// TIA Portal V20 export
FUNCTION_BLOCK "LER_LaserMark"   // FB9, LAD
// stored: Access Published, MemoryReserve 100, SetENOAutomatically false
   VAR_INPUT
      enable : Bool;
      enableManualCmds : Bool;
      jellyRollUsed : Bool;   // Unused is dryrun, gaugeRnR etc..
      simulationCmds : Bool;
      errAckHmi : Bool;
      interlock : Bool;
      autoGenMarkingData : String[32];
   END_VAR
   VAR_OUTPUT
      lagerMarkingTrigger : Bool;
      error : Bool;
      errorCode : Word;
   END_VAR
   VAR_IN_OUT
      configuration : "LER_typeLaserMarkConfiguration";
      moduleInterface : "LER_typeLaserMarkInterface";
      controlNode : "LER_typeLaserMarkControlNode";
   END_VAR
   VAR
      instTONTimer { S7_SetPoint := 'True'} : Array[0..19] of IEC_TIMER;
      statCmd { ExternalAccessible := 'False'; ExternalVisible := 'False'; ExternalWritable := 'False'} : "LER_typeLaserMarkCommands";
      statMonitoring { ExternalAccessible := 'False'; ExternalVisible := 'False'; ExternalWritable := 'False'} : "LER_typeLaserMarkMonitoring";
      statConfig { ExternalAccessible := 'False'; ExternalVisible := 'False'; ExternalWritable := 'False'} : "LER_typeLaserMarkConfiguration";
      statRetValInt { ExternalAccessible := 'False'; ExternalVisible := 'False'; ExternalWritable := 'False'} : Array[1..#count] of Int;
      statRetValWord { ExternalAccessible := 'False'; ExternalVisible := 'False'; ExternalWritable := 'False'} : Array[1..#count] of Word;
      statBit { ExternalAccessible := 'False'; ExternalVisible := 'False'; ExternalWritable := 'False'} : Array[0..49] of Bool;
      statAction { ExternalAccessible := 'False'; ExternalVisible := 'False'; ExternalWritable := 'False'} : Array[0..49] of Bool;
      statOutputCharData { ExternalAccessible := 'False'; ExternalVisible := 'False'; ExternalWritable := 'False'} : Array[1..128] of Char;
      statTpTimer { S7_SetPoint := 'True'} : Array[0..1] of TP_TIME;
      statPulse : Array[0..999] of Bool;
      statTonTimer { S7_SetPoint := 'True'} : Array[0..999] of TON_TIME;
      statProgramChange : Array[0..999] of Bool;
      "step" { ExternalAccessible := 'False'; ExternalVisible := 'False'; ExternalWritable := 'False'} : Int;
      statHold : Bool;
   END_VAR
   VAR_TEMP
      tempRetVal : Array[1..#count] of Int;
      tempCnt : Array[0..9] of UInt;
      tempCharDataDelete : Array[1..128] of Char;
      tempStringDataDelete : String[128];
      tempProgramNoDelete : DWord;
      tempIndex : Int;
   END_VAR
   VAR CONSTANT
      delayTime : Time := T#2s;
      count : Int := 16;
      statusNoErrorOccurred : Word := 16#0000;   // No error occurred.
      errMachine : Word := 16#8000;
      errRequest : Word := 16#8001;
      errHwdNotConfigured : Word := 16#8090;   // You have not configured a module for the specified hardware identifier or You have ignored the restriction concerning the length of consistent data, or you have not specified a hardware identifier as an address at parameter LADDR
      errRecordDataType : Word := 16#8092;   // Non-supported data type in the RECORD parameter.
      errNoDpProfinetIoModule : Word := 16#8093;   // No DP module/PROFINET IO device from which you can read consistent data exists for the hardware identifier specified in LADDR . This error code also occurs if the module addressed by means of LADDR does not have inputs.
      errIoAccessPermission : Word := 16#80A0;   // An access error was detected when accessing the I/O.
      errRecordLengthInsufficient : Word := 16#80B1;   // The length of the specified destination area at parameter RECORD is shorter than the configured user data length.
      errDataNotReceived : Word := 16#80C0;   // The data have not been read yet.
   END_VAR
   // // statBit[0] : data setting
   // // statBit[1] : delete data move
   // // statBit[2] : set data save
   // // statBit[3] : data write done
   // // statBit[4] : data writing
   // // statBit[5] : CMD_saveBT
   // // statBit[6] : CMD_save interlock
   // // statBit[7] : sequence hold
   // // statBit[8] : ( Not empty data ) read data save
   // // statBit[9] : ( Empty data ) read data save
   // // statBit[10] : write String To Char
   // // statBit[11] : done String To Char
   // // statBit[12] : P Trig
   // // statBit[15] : Temp config Save
   // // statBit[16] : config Save Lock
   // // statBit[17] : config Save Writing
   // // statBit[25] : trigger
   VAR_TEMP   // added for the SCL form of the ladder/FBD networks
      _w1 : Bool;
      _w2 : Bool;
      _w3 : Bool;
      _w4 : Bool;
      _w5 : Bool;
      _w6 : Bool;
      _w7 : Bool;
      _w8 : Bool;
      _w9 : Bool;
   END_VAR
BEGIN

REGION Network 1 (SCL): DP READ
   REGION DP read

       IF #enable AND NOT #simulationCmds THEN
           #"statRetValInt"[1] := DPRD_DAT(LADDR := #configuration.hwID.machineStatusID, RECORD => #statMonitoring.profinetInput.machineStatus);
           #"statRetValInt"[2] := DPRD_DAT(LADDR := #configuration.hwID.functionStatusID, RECORD => #statMonitoring.profinetInput.functionStatus);
           #"statRetValInt"[3] := DPRD_DAT(LADDR := #configuration.hwID.completionStatusID, RECORD => #statMonitoring.profinetInput.completionStatus);
           #"statRetValInt"[4] := DPRD_DAT(LADDR := #configuration.hwID.errorStatusID, RECORD => #statMonitoring.profinetInput.errorStatus);
           #"statRetValInt"[5] := DPRD_DAT(LADDR := #configuration.hwID.errorCodesID, RECORD => #statMonitoring.profinetInput.errorCodes);
           #"statRetValInt"[6] := DPRD_DAT(LADDR := #configuration.hwID.operateParameterID, RECORD => #statMonitoring.profinetInput.operateParameter);
           #"statRetValInt"[7] := DPRD_DAT(LADDR := #configuration.hwID."2DCReadResultID", RECORD => #statMonitoring.profinetInput."2DCReadResult");
           #"statRetValInt"[8] := DPRD_DAT(LADDR := #configuration.hwID.countResultDataID, RECORD => #statMonitoring.profinetInput.countResultData);
           #"statRetValInt"[9] := DPRD_DAT(LADDR := #configuration.hwID.resultDataID, RECORD => #statMonitoring.profinetInput.resultData);
       END_IF;

   END_REGION
END_REGION

REGION Network 2 (SCL): INPUT MAPPING
   REGION Input mapping

       IF #enable THEN
           // Command
           IF #enableManualCmds THEN
               #statCmd.start := #moduleInterface.commands.start;
               #statCmd.configSave := #moduleInterface.commands.configSave;
               #statMonitoring.profinetOutput.generalRequest.guideLaserRequest := #moduleInterface.commands.guideRequest;
               #statConfig.markingProgramNo := #moduleInterface.configuration.markingProgramNo;
           ELSE
               #statCmd.start := #controlNode.commands.start;
               #statCmd.configSave := #controlNode.commands.configSave;
               #statMonitoring.profinetOutput.generalRequest.guideLaserRequest := #controlNode.commands.guideRequest;
               #statConfig.markingProgramNo := #configuration.markingProgramNo;
           END_IF;

           #statCmd.generateMode := #moduleInterface.commands.generateMode;

           IF #statCmd.generateMode THEN
               #statConfig.markingData := #autoGenMarkingData;
           ELSE
               #statConfig.markingData := #moduleInterface.configuration.markingData;
           END_IF;

           #statMonitoring.data := #statConfig.markingData;

           #statMonitoring.error := #statMonitoring.profinetInput.machineStatus.errorStatus;
           #statMonitoring.warning := #statMonitoring.profinetInput.machineStatus.warningStatus;
           #statMonitoring.errorCode := #errorCode;

       END_IF;

   END_REGION
END_REGION

REGION Network 3 (SCL): ERROR STATUS
   REGION Error check

       IF #enable AND NOT #simulationCmds THEN
           IF #statRetValInt <> #tempRetVal THEN
               FOR #tempIndex := 1 TO #count DO
                   #statRetValWord[#tempIndex] := INT_TO_WORD(#statRetValInt[#tempIndex]); // convert the return value of DPRD, DPWR form int to word
                   CASE #statRetValWord[#tempIndex] OF

                       #errHwdNotConfigured:
                           #errorCode := #errHwdNotConfigured;

                       #errRecordDataType:
                           #errorCode := #errRecordDataType;

                       #errNoDpProfinetIoModule:
                           #errorCode := #errNoDpProfinetIoModule;

                       #errIoAccessPermission:
                           #errorCode := #errIoAccessPermission;

                       #errRecordLengthInsufficient:
                           #errorCode := #errRecordLengthInsufficient;

                       #errDataNotReceived:
                           #errorCode := #errDataNotReceived;
                   END_CASE;
               END_FOR;

           ELSIF #statMonitoring.profinetInput.machineStatus.errorStatus THEN
               #errorCode := #errMachine;

           ELSIF #statMonitoring.profinetInput.errorStatus.startMarkingRequestError OR
               #statMonitoring.profinetInput.errorStatus.stopMarkingRequestError OR
               #statMonitoring.profinetInput.errorStatus.errorClearRequestError OR
               #statMonitoring.profinetInput.errorStatus."2DCReadRequestError" OR
               #statMonitoring.profinetInput.errorStatus.commandSendRequestError THEN
               #errorCode := #errRequest;

           ELSE
               #errorCode := #statusNoErrorOccurred;
           END_IF;
       ELSE
           #errorCode := #statusNoErrorOccurred;
       END_IF;

       #error := #errorCode <> 0;

   END_REGION
END_REGION

REGION Network 4: ERROR ACK
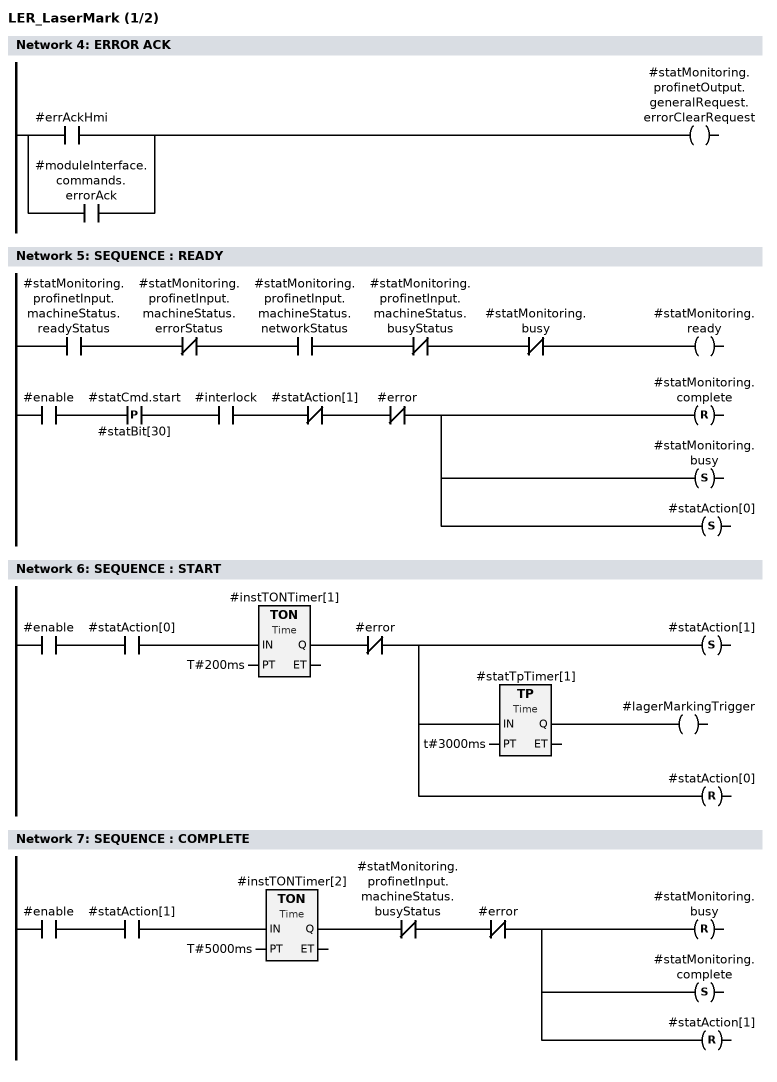
   RUNG wire#powerrail
      Contact( #errAckHmi )
      wire#w1
      Coil( #statMonitoring.profinetOutput.generalRequest.errorClearRequest )
   END_RUNG
   RUNG wire#powerrail
      Contact( #moduleInterface.commands.errorAck )
   END_RUNG wire#w1
   // the same network as SCL:
   #statMonitoring.profinetOutput.generalRequest.errorClearRequest := #errAckHmi OR #moduleInterface.commands.errorAck;
END_REGION

REGION Network 5: SEQUENCE : READY
   RUNG wire#powerrail
      Contact( #statMonitoring.profinetInput.machineStatus.readyStatus )
      I_Contact( #statMonitoring.profinetInput.machineStatus.errorStatus )
      Contact( #statMonitoring.profinetInput.machineStatus.networkStatus )
      I_Contact( #statMonitoring.profinetInput.machineStatus.busyStatus )
      I_Contact( #statMonitoring.busy )
      Coil( #statMonitoring.ready )
   END_RUNG
   RUNG wire#powerrail
      Contact( #enable )
      P_Contact(operand := #statCmd.start, bit := #statBit[30])
      Contact( #interlock )
      I_Contact( #statAction[1] )
      I_Contact( #error )
      wire#w1
      R_Coil( #statMonitoring.complete )
   END_RUNG
   RUNG wire#w1
      S_Coil( #statMonitoring.busy )
   END_RUNG
   RUNG wire#w1
      S_Coil( #statAction[0] )
   END_RUNG
   // the same network as SCL:
   #statMonitoring.ready := #statMonitoring.profinetInput.machineStatus.readyStatus AND NOT #statMonitoring.profinetInput.machineStatus.errorStatus AND #statMonitoring.profinetInput.machineStatus.networkStatus AND NOT #statMonitoring.profinetInput.machineStatus.busyStatus AND NOT #statMonitoring.busy;
   #_w1 := #enable AND #statCmd.start AND NOT #statBit[30];   // rising edge of #statCmd.start
   #statBit[30] := #statCmd.start;
   IF #_w1 AND #interlock AND NOT #statAction[1] AND NOT #error THEN
       #statMonitoring.complete := FALSE;
       #statMonitoring.busy := TRUE;
       #statAction[0] := TRUE;
   END_IF;
END_REGION

REGION Network 6: SEQUENCE : START
   RUNG wire#powerrail
      Contact( #enable )
      Contact( #statAction[0] )
      { S7_Templates := "time_type := Time" } #instTONTimer[1].TON(pt := T#200ms, et =>)
      I_Contact( #error )
      wire#w1
      S_Coil( #statAction[1] )
   END_RUNG
   RUNG wire#w1
      { S7_Templates := "time_type := Time" } #statTpTimer[1].TP(pt := t#3000ms, et =>)
      Coil( #lagerMarkingTrigger )
   END_RUNG
   RUNG wire#w1
      R_Coil( #statAction[0] )
   END_RUNG
   // the same network as SCL:
   #instTONTimer[1].TON(IN := #enable AND #statAction[0], PT := T#200ms);
   #_w1 := #instTONTimer[1].Q AND NOT #error;
   IF #_w1 THEN #statAction[1] := TRUE; END_IF;
   #statTpTimer[1].TP(IN := #_w1, PT := t#3000ms);
   #lagerMarkingTrigger := #statTpTimer[1].Q;
   IF #_w1 THEN #statAction[0] := FALSE; END_IF;
END_REGION

REGION Network 7: SEQUENCE : COMPLETE
   RUNG wire#powerrail
      Contact( #enable )
      Contact( #statAction[1] )
      { S7_Templates := "time_type := Time" } #instTONTimer[2].TON(pt := T#5000ms, et =>)
      I_Contact( #statMonitoring.profinetInput.machineStatus.busyStatus )
      I_Contact( #error )
      wire#w1
      R_Coil( #statMonitoring.busy )
   END_RUNG
   RUNG wire#w1
      S_Coil( #statMonitoring.complete )
   END_RUNG
   RUNG wire#w1
      R_Coil( #statAction[1] )
   END_RUNG
   // the same network as SCL:
   #instTONTimer[2].TON(IN := #enable AND #statAction[1], PT := T#5000ms);
   IF #instTONTimer[2].Q AND NOT #statMonitoring.profinetInput.machineStatus.busyStatus AND NOT #error THEN
       #statMonitoring.busy := FALSE;
       #statMonitoring.complete := TRUE;
       #statAction[1] := FALSE;
   END_IF;
END_REGION

REGION Network 8: CONFIGURATION
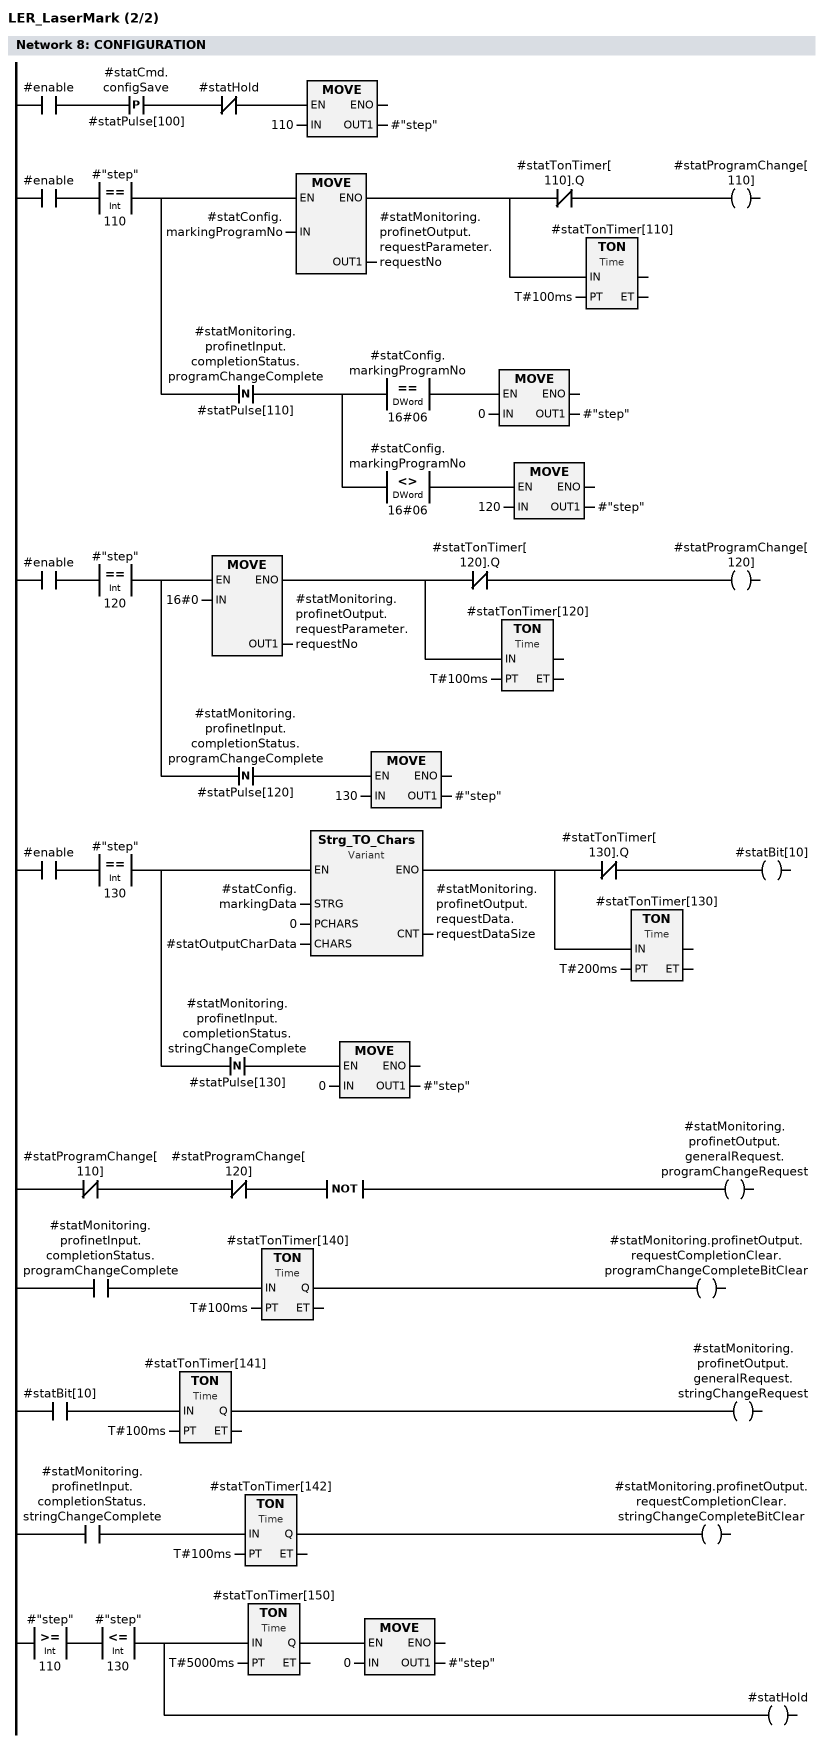
   RUNG wire#powerrail
      Contact( #enable )
      P_Contact(operand := #statCmd.configSave, bit := #statPulse[100])
      I_Contact( #statHold )
      Move(in := 110, out1 => #"step")
   END_RUNG
   RUNG wire#powerrail
      Contact( #enable )
      { S7_Templates := "SrcType := Int" } EQ_Contact(in1 := #"step", in2 := 110)
      wire#w1
      Move(in := #statConfig.markingProgramNo, out1 => #statMonitoring.profinetOutput.requestParameter.requestNo)
      wire#w2
      I_Contact( #statTonTimer[110].Q )
      Coil( #statProgramChange[110] )
   END_RUNG
   RUNG wire#w2
      { S7_Templates := "time_type := Time" } #statTonTimer[110].TON(pt := T#100ms, et =>)
   END_RUNG
   RUNG wire#w1
      N_Contact(operand := #statMonitoring.profinetInput.completionStatus.programChangeComplete, bit := #statPulse[110])
      wire#w3
      { S7_Templates := "SrcType := DWord" } EQ_Contact(in1 := #statConfig.markingProgramNo, in2 := 16#06)
      Move(in := 0, out1 => #"step")
   END_RUNG
   RUNG wire#w3
      { S7_Templates := "SrcType := DWord" } NE_Contact(in1 := #statConfig.markingProgramNo, in2 := 16#06)
      Move(in := 120, out1 => #"step")
   END_RUNG
   RUNG wire#powerrail
      Contact( #enable )
      { S7_Templates := "SrcType := Int" } EQ_Contact(in1 := #"step", in2 := 120)
      wire#w4
      Move(in := 16#0, out1 => #statMonitoring.profinetOutput.requestParameter.requestNo)
      wire#w5
      I_Contact( #statTonTimer[120].Q )
      Coil( #statProgramChange[120] )
   END_RUNG
   RUNG wire#w5
      { S7_Templates := "time_type := Time" } #statTonTimer[120].TON(pt := T#100ms, et =>)
   END_RUNG
   RUNG wire#w4
      N_Contact(operand := #statMonitoring.profinetInput.completionStatus.programChangeComplete, bit := #statPulse[120])
      Move(in := 130, out1 => #"step")
   END_RUNG
   RUNG wire#powerrail
      Contact( #enable )
      { S7_Templates := "SrcType := Int" } EQ_Contact(in1 := #"step", in2 := 130)
      wire#w6
      { S7_Templates := "[ptr_type := Variant, strg_type := String]" } Strg_TO_Chars(Strg := #statConfig.markingData, pChars := 0, Chars := #statOutputCharData, Cnt => #statMonitoring.profinetOutput.requestData.requestDataSize)
      wire#w7
      I_Contact( #statTonTimer[130].Q )
      Coil( #statBit[10] )
   END_RUNG
   RUNG wire#w7
      { S7_Templates := "time_type := Time" } #statTonTimer[130].TON(pt := T#200ms, et =>)
   END_RUNG
   RUNG wire#w6
      N_Contact(operand := #statMonitoring.profinetInput.completionStatus.stringChangeComplete, bit := #statPulse[130])
      Move(in := 0, out1 => #"step")
   END_RUNG
   RUNG wire#powerrail
      I_Contact( #statProgramChange[110] )
      I_Contact( #statProgramChange[120] )
      Not()
      Coil( #statMonitoring.profinetOutput.generalRequest.programChangeRequest )
   END_RUNG
   RUNG wire#powerrail
      Contact( #statMonitoring.profinetInput.completionStatus.programChangeComplete )
      { S7_Templates := "time_type := Time" } #statTonTimer[140].TON(pt := T#100ms, et =>)
      Coil( #statMonitoring.profinetOutput.requestCompletionClear.programChangeCompleteBitClear )
   END_RUNG
   RUNG wire#powerrail
      Contact( #statBit[10] )
      { S7_Templates := "time_type := Time" } #statTonTimer[141].TON(pt := T#100ms, et =>)
      Coil( #statMonitoring.profinetOutput.generalRequest.stringChangeRequest )
   END_RUNG
   RUNG wire#powerrail
      Contact( #statMonitoring.profinetInput.completionStatus.stringChangeComplete )
      { S7_Templates := "time_type := Time" } #statTonTimer[142].TON(pt := T#100ms, et =>)
      Coil( #statMonitoring.profinetOutput.requestCompletionClear.stringChangeCompleteBitClear )
   END_RUNG
   RUNG wire#powerrail
      { S7_Templates := "SrcType := Int" } GE_Contact(in1 := #"step", in2 := 110)
      { S7_Templates := "SrcType := Int" } LE_Contact(in1 := #"step", in2 := 130)
      wire#w8
      { S7_Templates := "time_type := Time" } #statTonTimer[150].TON(pt := T#5000ms, et =>)
      Move(in := 0, out1 => #"step")
   END_RUNG
   RUNG wire#w8
      Coil( #statHold )
   END_RUNG
   // the same network as SCL:
   #_w1 := #enable AND #statCmd.configSave AND NOT #statPulse[100];   // rising edge of #statCmd.configSave
   #statPulse[100] := #statCmd.configSave;
   IF #_w1 AND NOT #statHold THEN #"step" := 110; END_IF;
   #_w2 := #enable AND (#"step" = 110);
   IF #_w2 THEN
       #statMonitoring.profinetOutput.requestParameter.requestNo := #statConfig.markingProgramNo;
   END_IF;
   #statProgramChange[110] := #_w2 AND NOT #statTonTimer[110].Q;
   #statTonTimer[110].TON(IN := #_w2, PT := T#100ms);
   #_w3 := #_w2 AND NOT #statMonitoring.profinetInput.completionStatus.programChangeComplete AND #statPulse[110];   // falling edge of #statMonitoring.profinetInput.completionStatus.programChangeComplete
   #statPulse[110] := #statMonitoring.profinetInput.completionStatus.programChangeComplete;
   IF #_w3 AND (#statConfig.markingProgramNo = 16#06) THEN #"step" := 0; END_IF;
   IF #_w3 AND (#statConfig.markingProgramNo <> 16#06) THEN #"step" := 120; END_IF;
   #_w4 := #enable AND (#"step" = 120);
   IF #_w4 THEN #statMonitoring.profinetOutput.requestParameter.requestNo := 16#0; END_IF;
   #statProgramChange[120] := #_w4 AND NOT #statTonTimer[120].Q;
   #statTonTimer[120].TON(IN := #_w4, PT := T#100ms);
   #_w5 := #_w4 AND NOT #statMonitoring.profinetInput.completionStatus.programChangeComplete AND #statPulse[120];   // falling edge of #statMonitoring.profinetInput.completionStatus.programChangeComplete
   #statPulse[120] := #statMonitoring.profinetInput.completionStatus.programChangeComplete;
   IF #_w5 THEN #"step" := 130; END_IF;
   #_w6 := #enable AND (#"step" = 130);
   Strg_TO_Chars(EN := #_w6,
                 Strg := #statConfig.markingData,
                 pChars := 0,
                 Chars := #statOutputCharData,
                 Cnt => #statMonitoring.profinetOutput.requestData.requestDataSize,
                 ENO => #_w7);
   #statBit[10] := #_w7 AND NOT #statTonTimer[130].Q;
   #statTonTimer[130].TON(IN := #_w7, PT := T#200ms);
   #_w8 := #_w6 AND NOT #statMonitoring.profinetInput.completionStatus.stringChangeComplete AND #statPulse[130];   // falling edge of #statMonitoring.profinetInput.completionStatus.stringChangeComplete
   #statPulse[130] := #statMonitoring.profinetInput.completionStatus.stringChangeComplete;
   IF #_w8 THEN #"step" := 0; END_IF;
   #statMonitoring.profinetOutput.generalRequest.programChangeRequest := NOT (NOT #statProgramChange[110] AND NOT #statProgramChange[120]);
   #statTonTimer[140].TON(IN := #statMonitoring.profinetInput.completionStatus.programChangeComplete,
                          PT := T#100ms);
   #statMonitoring.profinetOutput.requestCompletionClear.programChangeCompleteBitClear := #statTonTimer[140].Q;
   #statTonTimer[141].TON(IN := #statBit[10], PT := T#100ms);
   #statMonitoring.profinetOutput.generalRequest.stringChangeRequest := #statTonTimer[141].Q;
   #statTonTimer[142].TON(IN := #statMonitoring.profinetInput.completionStatus.stringChangeComplete,
                          PT := T#100ms);
   #statMonitoring.profinetOutput.requestCompletionClear.stringChangeCompleteBitClear := #statTonTimer[142].Q;
   #_w9 := (#"step" >= 110) AND (#"step" <= 130);
   #statTonTimer[150].TON(IN := #_w9, PT := T#5000ms);
   IF #statTonTimer[150].Q THEN #"step" := 0; END_IF;
   #statHold := #_w9;
END_REGION

REGION Network 9 (SCL): REQUEST DATA
   IF #statBit[10] THEN
       #statMonitoring.profinetOutput.requestData.requestData1 := #statOutputCharData[1];
       #statMonitoring.profinetOutput.requestData.requestData2 := #statOutputCharData[2];
       #statMonitoring.profinetOutput.requestData.requestData3 := #statOutputCharData[3];
       #statMonitoring.profinetOutput.requestData.requestData4 := #statOutputCharData[4];
       #statMonitoring.profinetOutput.requestData.requestData5 := #statOutputCharData[5];
       #statMonitoring.profinetOutput.requestData.requestData6 := #statOutputCharData[6];
       #statMonitoring.profinetOutput.requestData.requestData7 := #statOutputCharData[7];
       #statMonitoring.profinetOutput.requestData.requestData8 := #statOutputCharData[8];
       #statMonitoring.profinetOutput.requestData.requestData9 := #statOutputCharData[9];

       #statMonitoring.profinetOutput.requestData.requestData10 := #statOutputCharData[10];
       #statMonitoring.profinetOutput.requestData.requestData11 := #statOutputCharData[11];
       #statMonitoring.profinetOutput.requestData.requestData12 := #statOutputCharData[12];
       #statMonitoring.profinetOutput.requestData.requestData13 := #statOutputCharData[13];
       #statMonitoring.profinetOutput.requestData.requestData14 := #statOutputCharData[14];
       #statMonitoring.profinetOutput.requestData.requestData15 := #statOutputCharData[15];
       #statMonitoring.profinetOutput.requestData.requestData16 := #statOutputCharData[16];
       #statMonitoring.profinetOutput.requestData.requestData17 := #statOutputCharData[17];
       #statMonitoring.profinetOutput.requestData.requestData18 := #statOutputCharData[18];
       #statMonitoring.profinetOutput.requestData.requestData19 := #statOutputCharData[19];

       #statMonitoring.profinetOutput.requestData.requestData20 := #statOutputCharData[20];
       #statMonitoring.profinetOutput.requestData.requestData21 := #statOutputCharData[21];
       #statMonitoring.profinetOutput.requestData.requestData22 := #statOutputCharData[22];
       #statMonitoring.profinetOutput.requestData.requestData23 := #statOutputCharData[23];
       #statMonitoring.profinetOutput.requestData.requestData24 := #statOutputCharData[24];
       #statMonitoring.profinetOutput.requestData.requestData25 := #statOutputCharData[25];
       #statMonitoring.profinetOutput.requestData.requestData26 := #statOutputCharData[26];
       #statMonitoring.profinetOutput.requestData.requestData27 := #statOutputCharData[27];
       #statMonitoring.profinetOutput.requestData.requestData28 := #statOutputCharData[28];
       #statMonitoring.profinetOutput.requestData.requestData29 := #statOutputCharData[29];

       #statMonitoring.profinetOutput.requestData.requestData30 := #statOutputCharData[30];
       #statMonitoring.profinetOutput.requestData.requestData31 := #statOutputCharData[31];
       #statMonitoring.profinetOutput.requestData.requestData32 := #statOutputCharData[32];
       #statMonitoring.profinetOutput.requestData.requestData33 := #statOutputCharData[33];
       #statMonitoring.profinetOutput.requestData.requestData34 := #statOutputCharData[34];
       #statMonitoring.profinetOutput.requestData.requestData35 := #statOutputCharData[35];
       #statMonitoring.profinetOutput.requestData.requestData36 := #statOutputCharData[36];
       #statMonitoring.profinetOutput.requestData.requestData37 := #statOutputCharData[37];
       #statMonitoring.profinetOutput.requestData.requestData38 := #statOutputCharData[38];
       #statMonitoring.profinetOutput.requestData.requestData39 := #statOutputCharData[39];

       #statMonitoring.profinetOutput.requestData.requestData40 := #statOutputCharData[40];
       #statMonitoring.profinetOutput.requestData.requestData41 := #statOutputCharData[41];
       #statMonitoring.profinetOutput.requestData.requestData42 := #statOutputCharData[42];
       #statMonitoring.profinetOutput.requestData.requestData43 := #statOutputCharData[43];
       #statMonitoring.profinetOutput.requestData.requestData44 := #statOutputCharData[44];
       #statMonitoring.profinetOutput.requestData.requestData45 := #statOutputCharData[45];
       #statMonitoring.profinetOutput.requestData.requestData46 := #statOutputCharData[46];
       #statMonitoring.profinetOutput.requestData.requestData47 := #statOutputCharData[47];
       #statMonitoring.profinetOutput.requestData.requestData48 := #statOutputCharData[48];
       #statMonitoring.profinetOutput.requestData.requestData49 := #statOutputCharData[49];

       #statMonitoring.profinetOutput.requestData.requestData50 := #statOutputCharData[50];
       #statMonitoring.profinetOutput.requestData.requestData51 := #statOutputCharData[51];
       #statMonitoring.profinetOutput.requestData.requestData52 := #statOutputCharData[52];
       #statMonitoring.profinetOutput.requestData.requestData53 := #statOutputCharData[53];
       #statMonitoring.profinetOutput.requestData.requestData54 := #statOutputCharData[54];
       #statMonitoring.profinetOutput.requestData.requestData55 := #statOutputCharData[55];
       #statMonitoring.profinetOutput.requestData.requestData56 := #statOutputCharData[56];
       #statMonitoring.profinetOutput.requestData.requestData57 := #statOutputCharData[57];
       #statMonitoring.profinetOutput.requestData.requestData58 := #statOutputCharData[58];
       #statMonitoring.profinetOutput.requestData.requestData59 := #statOutputCharData[59];

       #statMonitoring.profinetOutput.requestData.requestData60 := #statOutputCharData[60];
       #statMonitoring.profinetOutput.requestData.requestData61 := #statOutputCharData[61];
       #statMonitoring.profinetOutput.requestData.requestData62 := #statOutputCharData[62];
       #statMonitoring.profinetOutput.requestData.requestData63 := #statOutputCharData[63];
       #statMonitoring.profinetOutput.requestData.requestData64 := #statOutputCharData[64];
       #statMonitoring.profinetOutput.requestData.requestData65 := #statOutputCharData[65];
       #statMonitoring.profinetOutput.requestData.requestData66 := #statOutputCharData[66];
       #statMonitoring.profinetOutput.requestData.requestData67 := #statOutputCharData[67];
       #statMonitoring.profinetOutput.requestData.requestData68 := #statOutputCharData[68];
       #statMonitoring.profinetOutput.requestData.requestData69 := #statOutputCharData[69];

       #statMonitoring.profinetOutput.requestData.requestData70 := #statOutputCharData[70];
       #statMonitoring.profinetOutput.requestData.requestData71 := #statOutputCharData[71];
       #statMonitoring.profinetOutput.requestData.requestData72 := #statOutputCharData[72];
       #statMonitoring.profinetOutput.requestData.requestData73 := #statOutputCharData[73];
       #statMonitoring.profinetOutput.requestData.requestData74 := #statOutputCharData[74];
       #statMonitoring.profinetOutput.requestData.requestData75 := #statOutputCharData[75];
       #statMonitoring.profinetOutput.requestData.requestData76 := #statOutputCharData[76];
       #statMonitoring.profinetOutput.requestData.requestData77 := #statOutputCharData[77];
       #statMonitoring.profinetOutput.requestData.requestData78 := #statOutputCharData[78];
       #statMonitoring.profinetOutput.requestData.requestData79 := #statOutputCharData[79];

       #statMonitoring.profinetOutput.requestData.requestData80 := #statOutputCharData[80];
       #statMonitoring.profinetOutput.requestData.requestData81 := #statOutputCharData[81];
       #statMonitoring.profinetOutput.requestData.requestData82 := #statOutputCharData[82];
       #statMonitoring.profinetOutput.requestData.requestData83 := #statOutputCharData[83];
       #statMonitoring.profinetOutput.requestData.requestData84 := #statOutputCharData[84];
       #statMonitoring.profinetOutput.requestData.requestData85 := #statOutputCharData[85];
       #statMonitoring.profinetOutput.requestData.requestData86 := #statOutputCharData[86];
       #statMonitoring.profinetOutput.requestData.requestData87 := #statOutputCharData[87];
       #statMonitoring.profinetOutput.requestData.requestData88 := #statOutputCharData[88];
       #statMonitoring.profinetOutput.requestData.requestData89 := #statOutputCharData[89];

       #statMonitoring.profinetOutput.requestData.requestData90 := #statOutputCharData[90];
       #statMonitoring.profinetOutput.requestData.requestData91 := #statOutputCharData[91];
       #statMonitoring.profinetOutput.requestData.requestData92 := #statOutputCharData[92];
       #statMonitoring.profinetOutput.requestData.requestData93 := #statOutputCharData[93];
       #statMonitoring.profinetOutput.requestData.requestData94 := #statOutputCharData[94];
       #statMonitoring.profinetOutput.requestData.requestData95 := #statOutputCharData[95];
       #statMonitoring.profinetOutput.requestData.requestData96 := #statOutputCharData[96];
       #statMonitoring.profinetOutput.requestData.requestData97 := #statOutputCharData[97];
       #statMonitoring.profinetOutput.requestData.requestData98 := #statOutputCharData[98];
       #statMonitoring.profinetOutput.requestData.requestData99 := #statOutputCharData[99];

       #statMonitoring.profinetOutput.requestData.requestData100 := #statOutputCharData[100];
       #statMonitoring.profinetOutput.requestData.requestData101 := #statOutputCharData[101];
       #statMonitoring.profinetOutput.requestData.requestData102 := #statOutputCharData[102];
       #statMonitoring.profinetOutput.requestData.requestData103 := #statOutputCharData[103];
       #statMonitoring.profinetOutput.requestData.requestData104 := #statOutputCharData[104];
       #statMonitoring.profinetOutput.requestData.requestData105 := #statOutputCharData[105];
       #statMonitoring.profinetOutput.requestData.requestData106 := #statOutputCharData[106];
       #statMonitoring.profinetOutput.requestData.requestData107 := #statOutputCharData[107];
       #statMonitoring.profinetOutput.requestData.requestData108 := #statOutputCharData[108];
       #statMonitoring.profinetOutput.requestData.requestData109 := #statOutputCharData[109];

       #statMonitoring.profinetOutput.requestData.requestData110 := #statOutputCharData[110];
       #statMonitoring.profinetOutput.requestData.requestData111 := #statOutputCharData[111];
       #statMonitoring.profinetOutput.requestData.requestData112 := #statOutputCharData[112];
       #statMonitoring.profinetOutput.requestData.requestData113 := #statOutputCharData[113];
       #statMonitoring.profinetOutput.requestData.requestData114 := #statOutputCharData[114];
       #statMonitoring.profinetOutput.requestData.requestData115 := #statOutputCharData[115];
       #statMonitoring.profinetOutput.requestData.requestData116 := #statOutputCharData[116];
       #statMonitoring.profinetOutput.requestData.requestData117 := #statOutputCharData[117];
       #statMonitoring.profinetOutput.requestData.requestData118 := #statOutputCharData[118];
       #statMonitoring.profinetOutput.requestData.requestData119 := #statOutputCharData[119];

       #statMonitoring.profinetOutput.requestData.requestData120 := #statOutputCharData[120];
       #statMonitoring.profinetOutput.requestData.requestData121 := #statOutputCharData[121];
       #statMonitoring.profinetOutput.requestData.requestData122 := #statOutputCharData[122];
       #statMonitoring.profinetOutput.requestData.requestData123 := #statOutputCharData[123];
       #statMonitoring.profinetOutput.requestData.requestData124 := #statOutputCharData[124];
       #statMonitoring.profinetOutput.requestData.requestData125 := #statOutputCharData[125];
       #statMonitoring.profinetOutput.requestData.requestData126 := #statOutputCharData[126];
       #statMonitoring.profinetOutput.requestData.requestData127 := #statOutputCharData[127];
       #statMonitoring.profinetOutput.requestData.requestData128 := #statOutputCharData[128];
   END_IF;
END_REGION

REGION Network 10 (SCL): DP WRITE
   REGION DP write

       IF #enable AND NOT #simulationCmds THEN
           #"statRetValInt"[10] := DPWR_DAT(LADDR := #configuration.hwID.generalRequestID, RECORD := #statMonitoring.profinetOutput.generalRequest);
           #"statRetValInt"[11] := DPWR_DAT(LADDR := #configuration.hwID.functionRequestID, RECORD := #statMonitoring.profinetOutput.functionRequest);
           #"statRetValInt"[12] := DPWR_DAT(LADDR := #configuration.hwID.requestCompletionClearID, RECORD := #statMonitoring.profinetOutput.requestCompletionClear);
           #"statRetValInt"[13] := DPWR_DAT(LADDR := #configuration.hwID.requestParameterID, RECORD := #statMonitoring.profinetOutput.requestParameter);
           #"statRetValInt"[14] := DPWR_DAT(LADDR := #configuration.hwID.requestDataID, RECORD := #statMonitoring.profinetOutput.requestData);
       END_IF;

   END_REGION
END_REGION

REGION Network 11 (SCL): OUTPUT MAPPING
   REGION Output mapping
       //#statMonitoring.profinetOutput.generalRequest.startMarkingRequest := #statBit[25];
       #controlNode.commands.errorAck := #errAckHmi;
       //#moduleInterface.commands.errorAck := #errAckHmi;
       #controlNode.monitoring := #moduleInterface.monitoring := #statMonitoring;

   END_REGION
END_REGION
END_FUNCTION_BLOCK
